// TIA Portal V18 export
DATA_BLOCK "Debug"   // DB5
{ S7_Optimized_Access := 'TRUE' }
// stored: AutoNumber false, MemoryReserve 100
   VAR RETAIN
      SERVO_A1_LEGACY_MODE : Bool;
      SERVO_A2_LEGACY_MODE : Bool;
      SERVO_A3_LEGACY_MODE : Bool;
      SERVO_A4_LEGACY_MODE : Bool;
   END_VAR
   VAR
      "a3--start" : Bool;
   END_VAR
BEGIN
END_DATA_BLOCK
